# EPICS substitutions: iocs/example1/example1App/Db/template.substitutions
# My example template

file db/example.template { pattern
    { PREFIX,     SCAN }
    { $(pv_prefix) "1 second"}
    { $(pv_prefix) "3 second"}
}
